FUNCTION WRITE_PROTECTED_DATE_AND_TIME
VAR_INPUT
    Ptr : POINTER TO DATE_AND_TIME;
    Value : DATE_AND_TIME;
END_VAR

Ptr^ := Value;

END_FUNCTION

(* stored: Version 1.1.0.1, ProductVersion 3.1.4022.18
   POU WRITE_PROTECTED_DATE_AND_TIME: Id {af0064cc-fa42-4eeb-9659-37d82d6b5671}, SpecialFunc None *)
